{attribute addProperty BoxType "EK1100-0000-0018"}
{attribute addProperty Id "Beckhoff_ER7xxxEK1122Beckhoff_ER7xxxEK1122_C27AB41B2934366.75"}
{attribute addProperty CRC "2723724669"}
{attribute addProperty SizeInBites "2934"}
{attribute addProperty SizeInBytes "366.75"}
TYPE Beckhoff_ER7xxx_A258BD7D EXTENDS EK1100_179A0949 :
STRUCT
	{attribute addProperty Name "Beckhoff_ER7xxxEK1122"}
	Beckhoff_ER7xxxEK1122 : Beckhoff_ER7xxxEK1122_C27AB41B;
END_STRUCT
END_TYPE

(* stored: Version 1.2.0.0, ProductVersion 3.1.4024.9
   DUT Beckhoff_ER7xxx_A258BD7D: Id {265f333a-dc75-43c4-8ac7-6f3a88bb065b} *)
